{attribute addProperty BoxType "EK1122-0000-0018"}
{attribute addProperty Id "Beckhoff_EKx9xxsub_EK1100EK1100_179A0949162A_0001_EK1960_0000_0019EK1960_19ACB9CA59274A_0002_EK1960_0000_0021EK1960_B53F9B8356070A_0003_EK1960_0008_0019EK1960_19ACB9CA59274A_0004_EK1960_0008_0021EK1960_B53F9B8356070A_0005_EK1960_2600_0019EK1960_9C48564F59274A_0006_EK1960_2600_0021EK1960_4B393F5F59274A_0007_EK1960_2608_0019EK1960_9C48564F59274A_0008_EK1960_2608_0021EK1960_4B393F5F59274"}
{attribute addProperty CRC "577600848"}
{attribute addProperty SizeInBites "4688"}
{attribute addProperty SizeInBytes "586"}
TYPE Beckhoff_EKx9xxEK1122_226D7D50 EXTENDS EK1122_179A0949 :
STRUCT
	{attribute addProperty Name "Beckhoff_EKx9xxsub_EK1100"}
	Beckhoff_EKx9xxsub_EK1100 : EK1100_179A0949;
	{attribute addProperty Name "A_0001_EK1960_0000_0019"}
	A_0001_EK1960_0000_0019 : EK1960_19ACB9CA;
	{attribute addProperty Name "A_0002_EK1960_0000_0021"}
	A_0002_EK1960_0000_0021 : EK1960_B53F9B83;
	{attribute addProperty Name "A_0003_EK1960_0008_0019"}
	A_0003_EK1960_0008_0019 : EK1960_19ACB9CA;
	{attribute addProperty Name "A_0004_EK1960_0008_0021"}
	A_0004_EK1960_0008_0021 : EK1960_B53F9B83;
	{attribute addProperty Name "A_0005_EK1960_2600_0019"}
	A_0005_EK1960_2600_0019 : EK1960_9C48564F;
	{attribute addProperty Name "A_0006_EK1960_2600_0021"}
	A_0006_EK1960_2600_0021 : EK1960_4B393F5F;
	{attribute addProperty Name "A_0007_EK1960_2608_0019"}
	A_0007_EK1960_2608_0019 : EK1960_9C48564F;
	{attribute addProperty Name "A_0008_EK1960_2608_0021"}
	A_0008_EK1960_2608_0021 : EK1960_4B393F5F;
END_STRUCT
END_TYPE

(* stored: Version 1.2.0.0, ProductVersion 3.1.4024.9
   DUT Beckhoff_EKx9xxEK1122_226D7D50: Id {ba9646b7-5a62-4aa5-8f39-ec3b5187009e} *)
